TYPE ZCom :
STRUCT
  // module context
  App : ZApplication.ApplicationComPublish;
  Alarming : ZApplication.AlarmingCom;
  Messages : ZApplication.MessagingCom;
  
  // unit context
  Unit : ZComUnit;

END_STRUCT
END_TYPE

(* stored: Version 1.1.0.1
   DUT ZCom: Id {7aebe4cc-6a69-4d35-8fa5-f21343175150} *)
